// TwinCAT 3 PLC project Arrays1
// ProgramVersion: 3.1.4023.0
// libraries:
//   Tc2_Standard, * (Beckhoff Automation GmbH)
//   Tc2_System, * (Beckhoff Automation GmbH)
//   Tc3_Module, * (Beckhoff Automation GmbH)
// project tree:
//   / PlcTask.TcTTO
//   POUs/ MAIN.TcPOU
// real-time tasks:
//   TASK PlcTask: cycle T#10ms, priority 20, ADS port 350

CONFIGURATION Arrays1
    RESOURCE PLC ON TwinCAT3
        TASK PlcTask(INTERVAL := T#10ms, PRIORITY := 20);
        PROGRAM MAIN WITH PlcTask : MAIN;
    END_RESOURCE
END_CONFIGURATION

// ---- POUs/MAIN.TcPOU
PROGRAM MAIN
VAR
	aOneArray : ARRAY[1..5] OF INT := [4, 20, 30, 40, 50];
	nOneInt : INT;
END_VAR

aOneArray[1] := 42;
nOneInt := aOneArray[1] + aOneArray[4];

END_PROGRAM
